TYPE E_DayPhase :
(
    Morning,
    Noon,
    Evening,
    Night
);
END_TYPE

(* stored: Version 1.1.0.1, ProductVersion 3.1.4024.16
   DUT E_DayPhase: Id {68ee3359-0bc4-4fc3-9b3d-e09300f95794} *)
